TYPE ST_ScannerWriteData :
STRUCT
	TrigWrite	: BOOL; //temporary trigger for writing data
	Data		: T_MaxString := 'sRI0'; //sMN mTCgateon
	Busy		: BOOL;
END_STRUCT
END_TYPE

(* stored: Version 1.1.0.1, ProductVersion 3.1.4024.9
   DUT ST_ScannerWriteData: Id {fc5e5c15-cc19-4b13-a8c5-1eb8a0ff2f31} *)
